// TIA Portal V20 export
DATA_BLOCK "LBP_Axis02_Y"   // DB32
TITLE = Axis-specific signals
{ S7_Optimized_Access := 'FALSE' }
AUTHOR : SINUMERIK
FAMILY : SINUMERIK_ONE
VERSION : 6.14
// Interface between user program and axis/spindle, contains signals from/to axis/spindle 2
// stored: AutoNumber false, InstanceOfName LBP_typeAxisX, InstanceOfType UDT
"LBP_typeAxisX"
   // VAR RETAIN
   //    A_FD_OR : Byte;   // Feedrate override
   //    A_DriveEnable : Bool;   // Drive test movement enable
   //    A_AckFixedStop : Bool;   // Acknowledge fixed stop reached
   //    A_SensorFixedStop : Bool;   // Sensor fixed stop
   //    A_ASpDisable : Bool;   // Axis/spindle disable
   //    A_Follow_upMode : Bool;   // Follow-up mode
   //    A_PosMeas1 : Bool;   // Position measuring system 1
   //    A_PosMeas2 : Bool;   // Position measuring system 2
   //    A_ORactive : Bool;   // Override active
   //    A_SWCam : Bool;   // SW cam activation
   //    A_ContrEnable : Bool;   // Controller enable
   //    A_DelDTGSpReset : Bool;   // Delete distance to go/Spindle-Reset
   //    A_Clamp : Bool;   // Clamping in progress
   //    A_RefVal1 : Bool;   // Reference point value 1
   //    A_RefVal2 : Bool;   // Reference point value 2
   //    A_RefVal3 : Bool;   // Reference point value 3
   //    A_RefVal4 : Bool;   // Reference point value 4
   //    A_ExtZO : Bool;   // Import external ZO
   //    A_EnabTravFixedStop : Bool;   // Enable travel to fixed stop
   //    A_FixedFD1 : Bool;   // Activate fixed feed 1
   //    A_FixedFD2 : Bool;   // Activate fixed feed 2
   //    A_FixedFD3 : Bool;   // Activate fixed feed 3
   //    A_FixedFD4 : Bool;   // Activate fixed feed 4
   //    A_VelocSpeedLimit : Bool;   // Velocity/spindle speed limitation
   //    A_PrgtestAxRel : Bool;   // Program test axis/spindle release
   //    A_HW1 : Bool;   // Activate handwheel 1
   //    A_HW2 : Bool;   // Activate handwheel 2
   //    A_HW3 : Bool;   // Activate handwheel 3
   //    A_FDSpStop : Bool;   // Feed stop/spindle stop
   //    A_Disable : Bool;   // Traversing key disable
   //    A_RapidTrOR : Bool;   // Rapid traverse override
   //    A_Minus : Bool;   // Traversing key minus
   //    A_Plus : Bool;   // Traversing key plus
   //    A_INC1 : Bool;   // INC1
   //    A_INC10 : Bool;   // INC10
   //    A_INC100 : Bool;   // INC100
   //    A_INC1000 : Bool;   // INC1000
   //    A_INC10000 : Bool;   // INC10000
   //    A_INCVar : Bool;   // INC variable
   //    A_ContManTravel : Bool;   // Continuous manual travel
   //    f5_7 : Bool;
   //    A_OEMAxis : Byte;   // OEM axis signals
   //    A_InvHWDirOfRot : Bool;   // Inverting handwheel direction of rotation
   //    f7_1 : Bool;
   //    f7_2 : Bool;
   //    f7_3 : Bool;
   //    f7_4 : Bool;
   //    f7_5 : Bool;
   //    f7_6 : Bool;
   //    f7_7 : Bool;
   //    A_NCASpChanA : Bool;   // Assign NC axis/spindle channel A
   //    A_NCASpChanB : Bool;   // Assign NC axis/spindle channel B
   //    A_NCASpChanC : Bool;   // Assign NC axis/spindle channel C
   //    A_NCASpChanD : Bool;   // Assign NC axis/spindle channel D
   //    A_NCASpStrobe : Bool;   // Activation of assignment with pos. edge
   //    f8_5 : Bool;
   //    f8_6 : Bool;
   //    A_PLCASp : Bool;   // Request PLC axis/spindle
   //    A_Para_A : Bool;   // Parameter block servo A
   //    A_Para_B : Bool;   // Parameter block servo B
   //    A_Para_C : Bool;   // Parameter block servo C
   //    A_LockParSetDef : Bool;   // Lock parameter set definition from NC
   //    f9_4 : Bool;
   //    f9_5 : Bool;
   //    f9_6 : Bool;
   //    f9_7 : Bool;
   //    A_REPOSDelay : Bool;   // REPOS DELAY
   //    f10_1 : Bool;
   //    f10_2 : Bool;
   //    f10_3 : Bool;
   //    f10_4 : Bool;
   //    f10_5 : Bool;
   //    f10_6 : Bool;
   //    f10_7 : Bool;
   //    A_StartBrakeTest : Bool;   // Start brake test
   //    f11_1 : Bool;
   //    f11_2 : Bool;
   //    f11_3 : Bool;
   //    f11_4 : Bool;
   //    f11_5 : Bool;
   //    f11_6 : Bool;
   //    f11_7 : Bool;
   //    A_HWLimitMinus : Bool;   // Hardware limit switch minus
   //    A_HWLimitPlus : Bool;   // Hardware limit switch plus
   //    A_SWLimit2Minus : Bool;   // 2nd software limit switch minus
   //    A_SWLimit2Plus : Bool;   // 2nd software limit switch plus
   //    A_ModuloLimitEn : Bool;   // Modulo limit enabled
   //    f12_5 : Bool;
   //    f12_6 : Bool;
   //    A_DelayRef : Bool;   // Delay reference point approach
   //    A_JogFixPPos0 : Bool;   // JogFixPointPos 0
   //    A_JogFixPPos1 : Bool;   // JogFixPointPos 1
   //    A_JogFixPPos2 : Bool;   // JogFixPointPos 2
   //    A_JogToPos : Bool;   // Jog to position
   //    f13_4 : Bool;
   //    f13_5 : Bool;
   //    f13_6 : Bool;
   //    f13_7 : Bool;
   //    A_ProgtestSuppress : Bool;   // Program test to suppress
   //    A_ProgtestActivate : Bool;   // Program test activate
   //    f14_2 : Bool;
   //    f14_3 : Bool;
   //    f14_4 : Bool;
   //    f14_5 : Bool;
   //    f14_6 : Bool;
   //    f14_7 : Bool;
   //    f15 : Byte;
   //    A_ActGearA : Bool;   // Actual gear stage A
   //    A_ActGearB : Bool;   // Actual gear stage B
   //    A_ActGearC : Bool;   // Actual gear stage C
   //    A_GearChangeOv : Bool;   // Gear has changed over
   //    A_Sp1Syn : Bool;   // Re-synchronize spindle 1
   //    A_Sp2Syn : Bool;   // Re-synchronize spindle 2
   //    A_NoMonitorGear : Bool;   // No monitoring when changing gear
   //    A_DeleteS : Bool;   // Delete S value
   //    A_FD_ORSp : Bool;   // Feedrate override for spindle valid
   //    f17_1 : Bool;
   //    f17_2 : Bool;
   //    f17_3 : Bool;
   //    A_Sp1SynP : Bool;   // Re-synchronize spindle 1 for positioning
   //    A_Sp2SynP : Bool;   // Re-synchronize spindle 2 for positioning
   //    A_M3M4Inv : Bool;   // Invert M3/M4
   //    f17_7 : Bool;
   //    f18_0 : Bool;
   //    f18_1 : Bool;
   //    f18_2 : Bool;
   //    f18_3 : Bool;
   //    A_OscilPLC : Bool;   // Oscillation via PLC
   //    A_OscilSpeed : Bool;   // Enable Oscillation
   //    A_SetRotDirectRight : Bool;   // Setpoint osci. direct. right
   //    A_SetRotDirectLeft : Bool;   // Setpoint osci. direct. left
   //    A_SpOR : Byte;   // Spindle override
   //    f20_0 : Bool;
   //    A_RUEncQuStop : Bool;   // Run-up encoder quick stop
   //    f20_2 : Bool;
   //    A_SpeedSetpSmooth : Bool;   // Speed setpoint smoothing
   //    f20_4 : Bool;
   //    A_HoldBrakeToOpen : Bool;   // Holding brake open
   //    f20_6 : Bool;
   //    f20_7 : Bool;
   //    A_ParA : Bool;   // Parameter set selection A
   //    A_ParB : Bool;   // Parameter set selection B
   //    A_ParC : Bool;   // Parameter set selection C
   //    A_MotA : Bool;   // Motor selection A
   //    A_MotB : Bool;   // Motor selection B
   //    A_MotOK : Bool;   // Motor selected
   //    A_IntegratDisable : Bool;   // N controller integrator disable
   //    A_PulseEnable : Bool;   // Pulse enable
   //    f22_0 : Bool;
   //    f22_1 : Bool;
   //    f22_2 : Bool;
   //    f22_3 : Bool;
   //    f22_4 : Bool;
   //    f22_5 : Bool;
   //    f22_6 : Bool;
   //    f22_7 : Bool;
   //    f23_0 : Bool;
   //    f23_1 : Bool;
   //    f23_2 : Bool;
   //    f23_3 : Bool;
   //    f23_4 : Bool;
   //    f23_5 : Bool;
   //    f23_6 : Bool;
   //    f23_7 : Bool;
   //    f24_0 : Bool;
   //    A_ControlAx : Bool;   // Control Axis
   //    f24_2 : Bool;
   //    f24_3 : Bool;
   //    A_TorqComp : Bool;   // Torque compensation
   //    A_ChangSetpOutAss0 : Bool;   // Bit value for CTRLOUT_changed - Change setpoint output assignment
   //    A_ChangSetpOutAss1 : Bool;   // Bit value for CTRLOUT_changed - Change setpoint output assignment
   //    A_MS : Bool;   // Master / Slave On
   //    A_DynBComp : Bool;   // Dynamic backlash compensation activated
   //    f25_1 : Bool;
   //    f25_2 : Bool;
   //    f25_3 : Bool;
   //    f25_4 : Bool;
   //    f25_5 : Bool;
   //    f25_6 : Bool;
   //    f25_7 : Bool;
   //    f26_0 : Bool;
   //    f26_1 : Bool;
   //    f26_2 : Bool;
   //    A_CompContr : Bool;   // Compensation controller On
   //    A_FollowAxOv : Bool;   // Enable following axis override
   //    f26_5 : Bool;
   //    f26_6 : Bool;
   //    f26_7 : Bool;
   //    A_DEPMCS : Bool;   // Resume: DEPMCS
   //    A_DEPBCS : Bool;   // Resume: DEPBCS
   //    A_Corr : Bool;   // Resume: Corr
   //    A_HIAxMove : Bool;   // Resume: HIAxMove
   //    A_StopDEPMCS : Bool;   // Stop: DEPMCS
   //    A_StopDEPBCS : Bool;   // Stop: DEPBCS
   //    A_StopCorr : Bool;   // Stop: Corr
   //    A_StopHIAxMove : Bool;   // Stop: HIAxMove
   //    A_OscillAxExtRev : Bool;   // OscillAxExtReversal
   //    A_AxReset : Bool;   // AXRESET
   //    A_AxResume : Bool;   // AXRESUME
   //    A_SetRP : Bool;   // Set reversal point
   //    A_ChangeRP : Bool;   // Change reversal point
   //    A_StopRP : Bool;   // Stop at next reversal point
   //    A_Stop : Bool;   // Stop
   //    A_PLCAxis : Bool;   // PLC checks axis
   //    f29_0 : Bool;
   //    f29_1 : Bool;
   //    f29_2 : Bool;
   //    f29_3 : Bool;
   //    A_StartGantSynRun : Bool;   // Start gantry synchronization run
   //    A_NoAutoSync : Bool;   // No auto sync
   //    f29_6 : Bool;
   //    f29_7 : Bool;
   //    A_StopSpindle : Bool;   // Stop spindle
   //    A_StartCW : Bool;   // Start spindle clockwise
   //    A_StartCCW : Bool;   // Start spindle counterclockwise
   //    A_AutoGearStep : Bool;   // Autom. gear step change
   //    A_PosSpindle : Bool;   // Position spindle
   //    f30_5 : Bool;
   //    f30_6 : Bool;
   //    f30_7 : Bool;
   //    f31_0 : Bool;
   //    f31_1 : Bool;
   //    f31_2 : Bool;
   //    f31_3 : Bool;
   //    A_Resynchronize : Bool;   // Resynchronize
   //    A_DisSync : Bool;   // Disable synchronization
   //    A_Tracksync : Bool;   // Track synchronism
   //    A_DelSyncRunCorr : Bool;   // Deleting synchronous run correction
   //    f32_0 : Bool;
   //    f32_1 : Bool;
   //    f32_2 : Bool;
   //    f32_3 : Bool;
   //    f32_4 : Bool;
   //    f32_5 : Bool;
   //    f32_6 : Bool;
   //    f32_7 : Bool;
   //    f33_0 : Bool;
   //    f33_1 : Bool;
   //    f33_2 : Bool;
   //    f33_3 : Bool;
   //    f33_4 : Bool;
   //    f33_5 : Bool;
   //    f33_6 : Bool;
   //    f33_7 : Bool;
   //    A_SI_SetpLimBit0 : Bool;   // Set point limitation Bit0
   //    A_SI_SetpLimBit1 : Bool;   // Set point limitation Bit1
   //    f34_2 : Bool;
   //    A_ActivateBrakeRampForSs2e : Bool;
   //    f34_4 : Bool;
   //    f34_5 : Bool;
   //    f34_6 : Bool;
   //    f34_7 : Bool;
   //    f35 : Byte;
   //    f36 : Array[36..55] of Byte;
   //    A_FeedDriveCAxEng : Bool;   // Separate feed drive as C axis engaged
   //    A_SpSpeedDisp : Bool;   // Spindle speed display
   //    A_SpInsideClamp : Bool;   // Spindle inside clamping
   //    f56_3 : Bool;
   //    f56_4 : Bool;
   //    f56_5 : Bool;
   //    f56_6 : Bool;
   //    f56_7 : Bool;
   //    f57 : Byte;
   //    f58 : Word;
   //    E_SpNA : Bool;   // Spindle/no axis
   //    E_NCU_Link : Bool;   // NCU_link active axis
   //    E_EncodFreq1 : Bool;   // Encoder limit frequency 1 exceeded
   //    E_EncodFreq2 : Bool;   // Encoder limit frequency 2 exceeded
   //    E_RefSyn1 : Bool;   // Referenced/synchronized 1
   //    E_RefSyn2 : Bool;   // Referenced/synchronized 2
   //    E_ExactCoarse : Bool;   // Position reached with exact stop coarse
   //    E_ExactFine : Bool;   // Position reached with exact stop fine
   //    E_TravRequ : Bool;   // Travel request
   //    E_AxialAlarm : Bool;   // Axial alarm
   //    E_AxisReady : Bool;   // Axis ready
   //    E_Follow_upMode : Bool;   // Follow-up mode active
   //    E_Stat : Bool;   // Axis/spindle stationary (n<nmin)
   //    E_PositContr : Bool;   // Position controller active
   //    E_SpeedContr : Bool;   // Speed controller active
   //    E_CurrentContr : Bool;   // Current controller active
   //    E_SWCam : Bool;   // Software cams active
   //    E_HWOverlay : Bool;   // Handwheel overlay active
   //    E_RevFD : Bool;   // Revolutional feedrate active
   //    E_MeasAct : Bool;   // Measuring active
   //    E_ActTravFStop : Bool;   // Activate travel to fixed stop
   //    E_FixedStop : Bool;   // Fixed stop reached
   //    E_ForceFixedStop : Bool;   // Force fixed stop limited
   //    E_AxContainerRot : Bool;   // Axis container rotation active
   //    E_AxReset : Bool;   // Axis reset done
   //    E_PLCCtrlAx : Bool;   // PLC controlled axis
   //    E_AxStop : Bool;   // Axis stop active
   //    E_AxSpDisable : Bool;   // Axis/spindle disable active
   //    E_StopDEPMCS : Bool;   // Stop DEPMCS active
   //    E_StopDEPBCS : Bool;   // Stop DEPBCS active
   //    E_StopCorr : Bool;   // Stop Corr active
   //    E_StopHIAxMove : Bool;   // Stop HIAxMove active
   //    E_HW1 : Bool;   // Handwheel 1 active
   //    E_HW2 : Bool;   // Handwheel 2 active
   //    E_HW3 : Bool;   // Handwheel 3 active
   //    f64_3 : Bool;
   //    E_TReqMinus : Bool;   // Travel request minus
   //    E_TReqPlus : Bool;   // Travel request plus
   //    E_TCMinus : Bool;   // Traverse command minus
   //    E_TCPlus : Bool;   // Traverse command plus
   //    E_INC1 : Bool;   // INC1
   //    E_INC10 : Bool;   // INC10
   //    E_INC100 : Bool;   // INC100
   //    E_INC1000 : Bool;   // INC1000
   //    E_INC10000 : Bool;   // INC10000
   //    E_INCVar : Bool;   // INC variable
   //    E_ContManTravelAct : Bool;   // Continuous manual travel active
   //    f65_7 : Bool;
   //    E_OEMAxis : Byte;   // OEM axis signals
   //    E_InvHWDirOfRot : Bool;   // Handwheel direction of rotation invert actively
   //    f67_1 : Bool;
   //    f67_2 : Bool;
   //    f67_3 : Bool;
   //    f67_4 : Bool;
   //    f67_5 : Bool;
   //    f67_6 : Bool;
   //    f67_7 : Bool;
   //    E_NCASpChanA : Bool;   // NC axis/spindle in channel A
   //    E_NCASpChanB : Bool;   // NC axis/spindle in channel B
   //    E_NCASpChanC : Bool;   // NC axis/spindle in channel C
   //    E_NCASpChanD : Bool;   // NC axis/spindle in channel D
   //    E_PLCType : Bool;   // New type requested by PLC
   //    E_ChPoss : Bool;   // Change axis possible
   //    E_NeutrASp : Bool;   // Neutral axis/spindle
   //    E_PLCASp : Bool;   // PLC axis/spindle
   //    E_ParS_A : Bool;   // Parameter block servo A
   //    E_ParS_B : Bool;   // Parameter block servo B
   //    E_ParS_C : Bool;   // Parameter block servo C
   //    E_NCUNumLink_3 : Bool;
   //    E_NCUNumLink_4 : Bool;
   //    E_NCUNumLink_5 : Bool;
   //    E_NCUNumLink_6 : Bool;
   //    E_NCUNumLink_7 : Bool;
   //    E_ReposSh : Bool;   // REPOS shift
   //    E_ReposShValid : Bool;   // REPOS shift valid
   //    E_ReposDelayQuit : Bool;   // REPOS delay quit
   //    f70_3 : Bool;
   //    f70_4 : Bool;
   //    E_SI_Drv_SICSCC : Bool;   // DRV-Safety Integrated with SIC/SCC active
   //    E_SI_Drv_Parameterized : Bool;
   //    f70_7 : Bool;
   //    E_BrakeTest : Bool;   // Brake test active
   //    f71_1 : Bool;
   //    f71_2 : Bool;
   //    f71_3 : Bool;
   //    E_POS_RESTORED1 : Bool;   // POS_RESTORED 1
   //    E_POS_RESTORED2 : Bool;   // POS_RESTORED 2
   //    f71_6 : Bool;
   //    E_PLCAxDedic : Bool;   // PLC axis dedicated
   //    E_MMC_REPOSDelay : Bool;   // HMI REPOS DELAY
   //    f72_1 : Bool;
   //    f72_2 : Bool;
   //    f72_3 : Bool;
   //    f72_4 : Bool;
   //    f72_5 : Bool;
   //    f72_6 : Bool;
   //    f72_7 : Bool;
   //    f73 : Byte;
   //    f74_0 : Bool;
   //    f74_1 : Bool;
   //    f74_2 : Bool;
   //    f74_3 : Bool;
   //    E_ModLimEnAct : Bool;   // Modulo limit enabled active
   //    f74_5 : Bool;
   //    f74_6 : Bool;
   //    f74_7 : Bool;
   //    E_JogFixPPos0Act : Bool;   // JogFixPointPos 0 active
   //    E_JogFixPPos1Act : Bool;   // JogFixPointPos 1 active
   //    E_JogFixPPos2Act : Bool;   // JogFixPointPos 2 active
   //    E_JogFixPPos0 : Bool;   // JogFixPointPos 0 reached
   //    E_JogFixPPos1 : Bool;   // JogFixPointPos 1 reached
   //    E_JogFixPPos2 : Bool;   // JogFixPointPos 2 reached
   //    E_JogToPos : Bool;   // Jog to position active
   //    E_JogPos : Bool;   // Jog position reached
   //    E_ScratchPulse : Bool;   // Scratch pulse
   //    f76_1 : Bool;
   //    f76_2 : Bool;
   //    f76_3 : Bool;
   //    E_PathAxis : Bool;   // Path axis
   //    E_PosAxis : Bool;   // Positioning axis
   //    E_IndexAxisPos : Bool;   // Indexing axis in position
   //    E_CurvePos : Bool;   // Curve axis in position
   //    E_CollCheckRedSpeed : Bool;   // Reduced speed of Collisions Check
   //    f77_1 : Bool;
   //    f77_2 : Bool;
   //    f77_3 : Bool;
   //    f77_4 : Bool;
   //    f77_5 : Bool;
   //    f77_6 : Bool;
   //    f77_7 : Bool;
   //    E_FPosAxis : Real;   // F function (REAL format) for positioning axes
   //    E_SetpGearA : Bool;   // Setpoint gear stage A
   //    E_SetpGearB : Bool;   // Setpoint gear stage B
   //    E_SetpGearC : Bool;   // Setpoint gear stage C
   //    E_GearChange : Bool;   // Gear changeover
   //    f82_4 : Bool;
   //    f82_5 : Bool;
   //    f82_6 : Bool;
   //    f82_7 : Bool;
   //    E_SpeedLimit : Bool;   // Speed limit exceeded
   //    E_SetSpeedLimit : Bool;   // Setpoint speed limited
   //    E_SetSpeedIncreased : Bool;   // Setpoint speed increased
   //    E_GeoMonit : Bool;   // Geometry monitoring
   //    E_SupportAreaViol : Bool;   // Support area limits violated
   //    E_SetRange : Bool;   // Spindle in setpoint range
   //    E_SpeedMonit : Bool;   // Speed monitoring
   //    E_ActRotRight : Bool;   // Actual rotation direction right
   //    E_ConstCuttSpeed : Bool;   // Const. cutting speed active
   //    E_SUG : Bool;   // SUG active (grinding wheel surface speed)
   //    E_CLG : Bool;   // CLG active
   //    E_Tapping : Bool;   // Tapping without compensating chuck
   //    E_SyncMode : Bool;   // Synchronous mode spindle active
   //    E_PosMode : Bool;   // Positioning mode spindle active
   //    E_OscillMode : Bool;   // Oscillation mode spindle active
   //    E_ContrMode : Bool;   // Control mode spindle active
   //    E_ToolDynLimit : Bool;   // Tool with dynamics limit
   //    f85_1 : Bool;
   //    f85_2 : Bool;
   //    f85_3 : Bool;
   //    f85_4 : Bool;
   //    E_SpInPosition : Bool;   // Spindle in position
   //    f85_6 : Bool;
   //    f85_7 : Bool;
   //    E_MFunct : Int;   // M function (INT) for spindle
   //    E_SFunct : Real;   // S function (REAL) for spindle
   //    f92_0 : Bool;
   //    E_RUEncDisabl : Bool;   // Run-up encoder disable active
   //    f92_2 : Bool;
   //    E_SpeedSetpSmooth : Bool;   // Speed setpoint smoothing active
   //    E_RLIact : Bool;   // RLI active
   //    E_HoldBrakeOpened : Bool;   // Holding brake opened
   //    f92_6 : Bool;
   //    E_DriveRunEn : Bool;   // Drive run enabled
   //    E_ParA : Bool;   // Active parameter set A
   //    E_ParB : Bool;   // Active parameter set B
   //    E_ParC : Bool;   // Active parameter set C
   //    E_MotA : Bool;   // Active motor A
   //    E_MotB : Bool;   // Active motor B
   //    E_MotOK : Bool;   // Drive ready
   //    E_IntegratDisable : Bool;   // N controller integrator disabled
   //    E_PulseEnable : Bool;   // Pulses enabled
   //    E_MTempWarn : Bool;   // Prewarning motor temperature
   //    E_HTempWarn : Bool;   // Prewarning heat sink temperature
   //    E_RUComplete : Bool;   // Ramp-up complete
   //    E_MdMdx : Bool;   // Md<Mdx
   //    E_NactNmin : Bool;   // nact<nmin
   //    E_NactNx : Bool;   // nact<nx
   //    E_NactNset : Bool;   // nact=nset
   //    E_Message : Bool;   // Variable message function
   //    E_UDClessAlThreshold : Bool;   // UDC-link < alarm threshold
   //    E_DcVoltageAlarmAct : Bool;   // ESR: DC link voltage is below the specified minimum
   //    E_GeneratorOperationAct : Bool;   // ESR: generator operation is active
   //    E_SpeedBelowMin : Bool;   // ESR: actual speed is below specified minimum speed - axis is a generator axis
   //    E_Message2 : Bool;
   //    E_Message3 : Bool;
   //    f95_6 : Bool;
   //    E_I2TLimit : Bool;   // Power Section I2T limit
   //    f96_0 : Bool;
   //    E_AxisCtrl : Bool;   // Axis control active
   //    E_MSFine : Bool;   // Master/Slave fine
   //    E_MSCoarse : Bool;   // Master/Slave coarse
   //    E_MSCompContr : Bool;   // Master/Slave compensation controller activated
   //    E_BitValCtrlOutChang0 : Bool;   // Bit value for CTRLOUT_changed 0: Change setpoint output assignment
   //    E_BitValCtrlOutChang1 : Bool;   // Bit value for CTRLOUT_changed 1: Change setpoint output assignment
   //    E_MS : Bool;   // Master/Slave active
   //    f97 : Byte;
   //    E_SyncronFine : Bool;   // Synchronism fine
   //    E_SyncronCoarse : Bool;   // Synchronism coarse
   //    E_ActValCoupling : Bool;   // Actual value coupling
   //    f98_3 : Bool;
   //    E_OverlayMotion : Bool;   // Overlaid motion
   //    E_SWL : Bool;   // Speed warning limit reached
   //    E_AWL : Bool;   // Acceleration warning limit reached
   //    E_EmRetr : Bool;   // Emergency retraction active
   //    E_MasterSp : Bool;   // Master spindle
   //    E_SlaveSp : Bool;   // Slave spindle
   //    E_SyncRunCorrDOut : Bool;   // Synchronous run correction driven out
   //    E_AxisAccel : Bool;   // Axis accelerated
   //    E_Sync : Bool;   // Synchronization active
   //    E_MSR : Bool;   // Max. speed reached
   //    E_MAR : Bool;   // Max. acceleration reached
   //    f99_7 : Bool;
   //    f100_0 : Bool;
   //    f100_1 : Bool;
   //    E_OscillAxExtRev : Bool;   // OscillAxExt Reversal active
   //    E_StopOscill : Bool;   // Oscillation cannot start
   //    E_ErrorOscill : Bool;   // Error during oscillation
   //    E_SparkOut : Bool;   // Spark-out active
   //    E_OscillMotion : Bool;   // Oscillation motion active
   //    E_Oscill : Bool;   // Oscillation active
   //    f101_0 : Bool;
   //    f101_1 : Bool;
   //    E_GantCOLimit : Bool;   // Gantry cut-off limit exceeded
   //    E_GantWarn : Bool;   // Gantry warning limit exceeded
   //    E_SynRunStart : Bool;   // Synchronization run ready to start
   //    E_GantGroupSyn : Bool;   // Gantry grouping is synchronous
   //    E_GantLeadAxis : Bool;   // Gantry leading axis
   //    E_GantAxis : Bool;   // Gantry axis
   //    E_DynBComp : Bool;   // Dynamic backlash compensation activated
   //    f102_1 : Bool;
   //    f102_2 : Bool;
   //    E_ClampTolerance : Bool;   // Clamp tolerance exceeded
   //    f102_4 : Bool;
   //    E_PosMeas1 : Bool;   // Position measuring system 1 active
   //    E_PosMeas2 : Bool;   // Position measuring system 2 active
   //    f102_7 : Bool;
   //    E_SyncRunCorrIncl : Bool;   // Synchronous run correction is included
   //    f103_1 : Bool;
   //    f103_2 : Bool;
   //    f103_3 : Bool;
   //    E_Syncron2Fine : Bool;   // Synchronism fine
   //    E_Syncron2Coarse : Bool;   // Synchronism coarse
   //    f103_6 : Bool;
   //    f103_7 : Bool;
   //    E_AIAxis : Array[1..31] of Bool;   // Active infeed axis[1..31]
   //    f108_0 : Bool;
   //    f108_1 : Bool;
   //    f108_2 : Bool;
   //    f108_3 : Bool;
   //    f108_4 : Bool;
   //    f108_5 : Bool;
   //    f108_6 : Bool;
   //    f108_7 : Bool;
   //    f109_0 : Bool;
   //    f109_1 : Bool;
   //    f109_2 : Bool;
   //    f109_3 : Bool;
   //    f109_4 : Bool;
   //    f109_5 : Bool;
   //    f109_6 : Bool;
   //    f109_7 : Bool;
   //    f110_0 : Bool;
   //    f110_1 : Bool;
   //    f110_2 : Bool;
   //    f110_3 : Bool;
   //    f110_4 : Bool;
   //    f110_5 : Bool;
   //    f110_6 : Bool;
   //    f110_7 : Bool;
   //    f111_0 : Bool;
   //    f111_1 : Bool;
   //    f111_2 : Bool;
   //    f111_3 : Bool;
   //    f111_4 : Bool;
   //    f111_5 : Bool;
   //    f111_6 : Bool;
   //    f111_7 : Bool;
   //    f112 : Byte;
   //    f113 : Byte;
   //    f114 : Byte;
   //    f115 : Byte;
   //    f116 : Byte;
   //    f117_0 : Bool;
   //    f117_1 : Bool;
   //    f117_2 : Bool;
   //    f117_3 : Bool;
   //    f117_4 : Bool;
   //    f117_5 : Bool;
   //    f117_6 : Bool;
   //    f117_7 : Bool;
   //    f118 : DWord;
   //    f122 : DWord;
   //    f126 : Word;   // Internal
   //    E_MMC_ProgtestSuppress : Bool;   // HMI->PLC: Suppress program test
   //    E_MMC_ProgtestActivate : Bool;   // HMI->PLC: Activate program test
   //    f128_2 : Bool;
   //    f128_3 : Bool;
   //    f128_4 : Bool;
   //    f128_5 : Bool;
   //    f128_6 : Bool;
   //    f128_7 : Bool;
   //    f129 : Byte;
   //    E_FormatBit0DDS : Bool;
   //    E_FormatBit1DDS : Bool;
   //    E_FormatBit2DDS : Bool;
   //    E_FormatBit3DDS : Bool;
   //    E_FormatBit4DDS : Bool;
   //    f130_5 : Bool;
   //    f130_6 : Bool;
   //    E_MDS_DDS_InterfacesValid : Bool;
   //    f131 : Byte;
   //    E_SensorAv : Bool;   // Sensors available
   //    E_S1aMeasARod : Bool;   // Sensor S1: analogous measurement position of actuating rod
   //    f132_2 : Bool;
   //    f132_3 : Bool;
   //    E_S4dPistonStopP : Bool;   // Sensor S4: digital value piston stop position
   //    E_S5dAngleShaft : Bool;   // Sensor S5: digital value angle situation shaft
   //    E_S6Temp : Bool;   // Sensor S6: temperature
   //    f132_7 : Bool;
   //    f133 : Byte;
   //    E_ClampingState : Int;   // State of the clamping system
   //    E_AnalogSensor : Int;   // Analog sensor on the motor
   //    f138_0 : Bool;
   //    f138_1 : Bool;
   //    f138_2 : Bool;
   //    f138_3 : Bool;
   //    E_S4PistonStopP : Bool;   // Sensor S4: piston stop position
   //    E_S5AngleShaft : Bool;   // Sensor S5: angle situation shaft
   //    f138_6 : Bool;
   //    f138_7 : Bool;
   //    f139 : Byte;
   //    SCC : Struct   // PLC to Drive (SCC)
   //       CW1 : Struct
   //          TeststopStart : Bool;   // Test stops for extended functions
   //          res140_1 : Bool;
   //          res140_2 : Bool;
   //          res140_3 : Bool;
   //          res140_4 : Bool;
   //          CloseBrake : Bool;   // Close internal Brake
   //          res140_6 : Bool;
   //          res140_7 : Bool;
   //          res141 : Byte;
   //       END_STRUCT;
   //       CW3 : Struct
   //          res142 : Byte;
   //          SelectionSBT : Bool;   // Selection: safe brake test
   //          BT_Start : Bool;   // Start: brake test
   //          Brake_1_2 : Bool;   // Brake test with brake 1 or 2
   //          DirOfROT : Bool;   // Direction of rotation
   //          Testseq_1_2 : Bool;   // Test sequence 1 or 2
   //          BrakeClosed : Bool;   // Feedback external brake
   //          res143_6 : Bool;
   //          res143_7 : Bool;
   //       END_STRUCT;
   //    END_STRUCT;
   //    res144_163 : Array[144..163] of Byte;
   //    SIC : Struct   // Drive to PLC (SIC)
   //       SW1 : Struct
   //          SLA_Sel : Bool;   // Safely Limited Acceleration selected
   //          SLS_LimBit0_Sel : Bool;   // Safely-Limited Speed: limit Bit0 selected
   //          SLS_LimBit1_Sel : Bool;   // Safely-Limited Speed: limit Bit1 selected
   //          res164_3 : Bool;
   //          res164_4 : Bool;
   //          res164_5 : Bool;
   //          ESR_Req : Bool;   // Extended Stop and Retract requested
   //          SF_Message_Act : Bool;   // Safety error active
   //          STO_Act : Bool;   // Safe torque off: active
   //          SS1_Act : Bool;   // Safe Stop1: active
   //          SS2_Act : Bool;   // Safe Stop2: active
   //          SOS_Act : Bool;   // Safe Operating Stop: active
   //          SLS_Act : Bool;   // Safely-Limited Speed: active
   //          SOS_Sel : Bool;   // Safe Operating Stop: selected
   //          SLS_Sel : Bool;   // Safely-Limited Speed: selected
   //          InternalEvent : Bool;   // Safety error with Stop A active
   //       END_STRUCT;
   //       SW2 : Struct
   //          SDI_P_Sel : Bool;   // Safe direction positive: selected
   //          SDI_N_Sel : Bool;   // Safe direction negative: selected
   //          res166_2 : Bool;
   //          res166_3 : Bool;
   //          TestStopAct : Bool;   // Test stop active
   //          TestStopReq : Bool;   // Test stop requested
   //          res166_6 : Bool;
   //          res166_7 : Bool;
   //          res167_0 : Bool;
   //          res167_1 : Bool;
   //          res167_2 : Bool;
   //          res167_3 : Bool;
   //          SLP_LimBit0_Sel : Bool;   // Safely-Limited Position: limit Bit0 selected
   //          res167_5 : Bool;
   //          res167_6 : Bool;
   //          SLP_Sel : Bool;   // Safely-Limited Position: selected
   //       END_STRUCT;
   //       V_Limit_B : DInt;   // Setpoint speed limit effective
   //       SW3 : Struct
   //          res172_0 : Bool;
   //          res172_1 : Bool;
   //          res172_2 : Bool;
   //          SS2E_ACTIVE : Bool;   // SS2E active
   //          SS2ESR : Bool;   // SS2ESR active
   //          res172_5 : Bool;
   //          AcceptSLPAct : Bool;   // Acceptance test Safely-Limited Position active
   //          AcceptTestSel : Bool;   // Acceptance test selected
   //          SBT_Sel : Bool;   // Safety break test: selected
   //          SetpSettingDrive : Bool;   // Setpoint input is in the drive during the SBT
   //          Brake_1_2 : Bool;   // Test with brake 1 or 2
   //          BT_Act : Bool;   // Brake test: active
   //          BT_OK : Bool;   // Brake test: OK
   //          BT_Finished : Bool;   // Brake test: finished
   //          BrakeReq : Bool;   // External brake close requested
   //          SignLoadTorque : Bool;   // Sign of load torque is negative
   //       END_STRUCT;
   //    END_STRUCT;
   //    res174_187 : Array[174..187] of Byte;
   //    CW7 : Struct
   //       ReservedBit08 : Bool;
   //       ReservedBit09 : Bool;
   //       ReservedBit10 : Bool;
   //       ReservedBit11 : Bool;
   //       ReservedBit12 : Bool;
   //       ReservedBit13 : Bool;
   //       ReservedBit14 : Bool;
   //       ReservedBit15 : Bool;
   //       A_DisablePowerReduction : Bool;   // DYNEGMA: disable power reduction
   //       A_DisableCurrReduction : Bool;   // Motor overtemperature: disable current reduction
   //       ReservedBit02 : Bool;
   //       ReservedBit03 : Bool;
   //       ReservedBit04 : Bool;
   //       ReservedBit05 : Bool;
   //       ReservedBit06 : Bool;
   //       ReservedBit07 : Bool;
   //    END_STRUCT;
   //    SW7 : Struct
   //       E_EncMaintenanceRequired : Bool;   // Encoder maintenance required
   //       ReservedBit09 : Bool;
   //       ReservedBit10 : Bool;
   //       ReservedBit11 : Bool;
   //       ReservedBit12 : Bool;
   //       ReservedBit13 : Bool;
   //       ReservedBit14 : Bool;
   //       ReservedBit15 : Bool;
   //       E_TorqueLimited : Bool;   // DYNEGMA: torque limited
   //       E_CurrReductionActive : Bool;   // Motor overtemperature: current reduction active
   //       E_MotorTempModelAlarm : Bool;   // Motor overtemperature: motor temperature model alarm active
   //       E_PolePosIdentPassed : Bool;   // Pole position identification with encoder successfully carried out
   //       ReservedBit04 : Bool;
   //       ReservedBit05 : Bool;
   //       E_AndConditionFulfilled : Bool;   // AND logic operation: condition fulfilled
   //       E_OrConditionFulfilled : Bool;   // OR logic operation: condition fulfilled
   //    END_STRUCT;
   // END_VAR
BEGIN
END_DATA_BLOCK
